FUNCTION_BLOCK FB_Ciecie_Komunikacja EXTENDS FB_LogowanieBledow_ElementZlozony
VAR_INPUT
END_VAR
VAR_OUTPUT
END_VAR
VAR
END_VAR

METHOD DefinicjaTabeliZdarzen_1031_Niemiecki : BOOL
VAR_INPUT
	arrTablicaDefinicjiZdarzenOpis			: REFERENCE TO ARRAY [1..GVL_LogowanieBledow_Stale.MAX_ILOSC_ZDARZEN] OF DUT_LogowanieBledow_ZdarzenieOpis;

END_VAR
//arrTablicaDefinicjiZdarzenOpis [iStartId+0].sOpis	:= 'DE - TESTOWA WIADOMOSC';
END_METHOD

METHOD DefinicjaTabeliZdarzen_1033_Angielski : BOOL
VAR_INPUT
	arrTablicaDefinicjiZdarzenOpis			: REFERENCE TO ARRAY [1..GVL_LogowanieBledow_Stale.MAX_ILOSC_ZDARZEN] OF DUT_LogowanieBledow_ZdarzenieOpis;

END_VAR
//arrTablicaDefinicjiZdarzenOpis [iStartId+0].sOpis	:= 'EN - TESTOWA WIADOMOSC';
END_METHOD

METHOD DefinicjaTabeliZdarzen_1045_Polski : BOOL
VAR_INPUT
	arrTablicaDefinicjiZdarzenOpis			: REFERENCE TO ARRAY [1..GVL_LogowanieBledow_Stale.MAX_ILOSC_ZDARZEN] OF DUT_LogowanieBledow_ZdarzenieOpis;

END_VAR
//arrTablicaDefinicjiZdarzenOpis [iStartId+0].sOpis	:= 'PL - TESTOWA WIADOMOSC';
END_METHOD

METHOD DefinicjaTabeliZdarzen_Ogolna : BOOL
VAR_INPUT
	arrTablicaDefinicjiZdarzen				: REFERENCE TO ARRAY [1..GVL_LogowanieBledow_Stale.MAX_ILOSC_ZDARZEN] OF DUT_LogowanieBledow_Zdarzenie;
	arrTablicaDefinicjiZdarzenOpis			: REFERENCE TO ARRAY [1..GVL_LogowanieBledow_Stale.MAX_ILOSC_ZDARZEN] OF DUT_LogowanieBledow_ZdarzenieOpis;
	arrTablicaDefinicjiZdarzenStan			: REFERENCE TO ARRAY [1..GVL_LogowanieBledow_Stale.MAX_ILOSC_ZDARZEN] OF DUT_LogowanieBledow_ZdarzenieStan;

	iIdZdarzenia							: REFERENCE TO INT;
	iNrPodzespolu							: INT := 0;
	iNrPodelementu							: INT := 0;
	iNrElementu								: INT := 0;
END_VAR
(*
//testowy blad
	iIdZdarzenia												:= iIdZdarzenia + 1;
	arrTablicaDefinicjiZdarzen [iIdZdarzenia].iIdZdarzenia		:= iIdZdarzenia;
	arrTablicaDefinicjiZdarzen [iIdZdarzenia].byRodzajZdarzenia	:= 3;
	arrTablicaDefinicjiZdarzen [iIdZdarzenia].sKodBledu			:= '0001';
	arrTablicaDefinicjiZdarzen [iIdZdarzenia].sNrKomponentu		:= GenerujNrKomponentu (iNrPodzespolu := iNrPodzespolu, iNrPodelementu := iNrPodelementu, iNrElementu := iNrElementu); 
	arrTablicaDefinicjiZdarzenOpis [iIdZdarzenia].iIdZdarzenia 	:= iIdZdarzenia;
	arrTablicaDefinicjiZdarzenStan [iIdZdarzenia].iIdZdarzenia 	:= iIdZdarzenia;
	arrTablicaDefinicjiZdarzenStan [iIdZdarzenia].bAktywne		:= FALSE;
	*)
END_METHOD

END_FUNCTION_BLOCK

(* stored: Version 1.1.0.1, ProductVersion 3.1.4024.11
   POU FB_Ciecie_Komunikacja: Id {66655f0f-bc68-429c-806b-696162ed7efd}, SpecialFunc None
   Method DefinicjaTabeliZdarzen_1031_Niemiecki: Id {974c9778-595f-4035-ae9c-68bce23fac46}
   Method DefinicjaTabeliZdarzen_1033_Angielski: Id {8cb1b9d2-f1a4-4c44-9e9a-1e08522260bf}
   Method DefinicjaTabeliZdarzen_1045_Polski: Id {8b261a8b-fa25-4dd9-9b48-535e6834c7a9}
   Method DefinicjaTabeliZdarzen_Ogolna: Id {2c88d539-4c63-43e9-b6b1-b1f538965c6c} *)
